{attribute addProperty BoxType "EK1122-0000-0018"}
{attribute addProperty Id "Beckhoff_CUxxxxsub_EK1100EK1100_179A0949162A_0001_CU1123_0000_0016A_0001_CU1123_0000_0016_A8E4CC63950118.75"}
{attribute addProperty CRC "2156194550"}
{attribute addProperty SizeInBites "966"}
{attribute addProperty SizeInBytes "120.75"}
TYPE Beckhoff_CUxxxxEK1122_8084EAF6 EXTENDS EK1122_179A0949 :
STRUCT
	{attribute addProperty Name "Beckhoff_CUxxxxsub_EK1100"}
	Beckhoff_CUxxxxsub_EK1100 : EK1100_179A0949;
	{attribute addProperty Name "A_0001_CU1123_0000_0016"}
	A_0001_CU1123_0000_0016 : A_0001_CU1123_0000_0016_A8E4CC63;
END_STRUCT
END_TYPE

(* stored: Version 1.2.0.0, ProductVersion 3.1.4024.9
   DUT Beckhoff_CUxxxxEK1122_8084EAF6: Id {5427eb77-61e4-4e3f-bd44-4bfa9461d650} *)
